// TwinCAT 3 PLC project Builder1
// ProgramVersion: 3.1.4023.0
// libraries:
//   Tc2_Standard, * (Beckhoff Automation GmbH)
//   Tc2_System, * (Beckhoff Automation GmbH)
//   Tc3_Module, * (Beckhoff Automation GmbH)
//   VisuSymbols,3.5.10.0,System
// project tree:
//   / Class Diagram.TcCD (not stored), ConcreteBuilder.TcPOU, Director.TcPOU, GlobalTextList.TcGTLO, ITF_Builder.TcIO, PlcTask.TcTTO, Product.TcPOU, Visualization Manager.TcVMO (not stored)
//   POUs/ MAIN.TcPOU
//   VISUs/ Visualization.TcVIS
// real-time tasks:
//   TASK PlcTask: cycle T#10ms, priority 20, ADS port 350

CONFIGURATION Builder1
    RESOURCE PLC ON TwinCAT3
        TASK PlcTask(INTERVAL := T#10ms, PRIORITY := 20);
        PROGRAM MAIN WITH PlcTask : MAIN;
    END_RESOURCE
END_CONFIGURATION

// ---- ITF_Builder.TcIO
///Builder interface to declare all needed parts to be built
INTERFACE ITF_Builder

///Illustrative method of the pattern to set the main part
METHOD Set_Main_Part
VAR_INPUT
	///Illustrative value (object because it is a TRING) to be set as a product part
	mainPart: STRING;
END_VAR
END_METHOD

///Illustrative method of the pattern to set the part1
METHOD Set_Part1
VAR_INPUT
	///Illustrative value (object because it is a TRING) to be set as a product part
	part1: STRING;
END_VAR
END_METHOD

///Illustrative method of the pattern to set the part2
METHOD Set_Part2
VAR_INPUT
	///Illustrative value (object because it is a TRING) to be set as a product part
	part2: STRING;
END_VAR
END_METHOD

///Illustrative method of the pattern to set the part3
METHOD Set_Part3
VAR_INPUT
	///Illustrative value (object because it is a TRING) to be set as a product part
	part3: STRING;
END_VAR
END_METHOD

END_INTERFACE

// ---- POUs/MAIN.TcPOU
PROGRAM MAIN
VAR
	///Three specifications arrays to be used by the same Director
	specsBuilder1: ARRAY[1..4] OF STRING := ['Red Chassis ', 'Sedan ', 'Motor 1.4cc ', 'Aluminium tires'];
	specsBuilder2: ARRAY[1..4] OF STRING := ['Black Chassis ', 'Hatchback ', 'Motor 2.0cc ', 'Chrome plated tires'];
	specsBuilder3: ARRAY[1..4] OF STRING := ['White Chassis ', 'Sport ', 'Motor 2.5cc ', 'Ligth aluminium tires'];
	///Special array for the visualization element
	tableArray: ARRAY[1..4, 1..3] OF STRING := ['Red Chassis', 'Black Chassis', 'White Chassis', 'Sedan', 'Hatchback', 'Sport', 'Motor 1.4cc', 'Motor 2.0cc', 'Motor 2.5cc', 'Aluminium tires', 'Chrome plated tires', 'Ligth aluminium tires'];
	///String variable to interact and respond to the client in the visualization element
	sMessageLog: STRING(500) := 'Waiting for your request';
	///Boolean value to react to a clients request
	bRequest: BOOL := FALSE;
	///Boolean and integer values to receive data from the tables in the visualization element
	///The boolean value validates if the client has chosen a valid option
	bRow: BOOL := FALSE;
	///The integer value hold the reference to the array of specifications
	iRow: INT := 0;
	///A pointer to Poduct to dynamically create and delete product objects at the clients requests
	prod: POINTER TO Product;
	///Three ConcreteBuilder instances to be passed to the Director and build the final Product objects
	///Each ConcreteBuilder intance is initiated with its own specifications
	{attribute 'old_input_assignments' := ''}
	concreteBuilder1: ConcreteBuilder(specs := specsBuilder1);
	{attribute 'old_input_assignments' := ''}
	concreteBuilder2: ConcreteBuilder(specs := specsBuilder2);
	{attribute 'old_input_assignments' := ''}
	concreteBuilder3: ConcreteBuilder(specs := specsBuilder3);
	///A Director instance that is instanciated with a ConcreteBuilder instance.
	/// later on in the program the specific ConcreteBuilder instance could be changed dynamically
	{attribute 'old_input_assignments' := ''}
	aDirector: Director(inputConcreteBuilder := concreteBuilder1);	
END_VAR

//The visualization element lets the client chose an option blueprint to build a Car
//Once the client has chosen his prefered option, he can then procede to make the request of construction.
//The bottom rectangle will handle all possible responses from te application to the client.

//If the client makes a request in the visualization element
IF bRequest
	THEN
	//CASE instruction to handle all possible cases of the cleint's request
	//The value to verify is iRow to specify which row the client has chosen
	CASE iRow OF
		//If the client has chosen the "Title" row from the visualization element we notify the client to chose a Car blueprint
		0: 	sMessageLog := 'You must first select a Car to make a request. Waiting for your request';
			//Once this reques has been handled, the reques flag is set to FALSE
			bRequest := FALSE;
		
		//If the client has chosen the first option row, the builder notifies the client about the received request
		1:	sMessageLog := 'Your red car is being built';
			//A new product object is created on demand
			prod := __NEW(Product);
			//The director object receives the ConcreteBuilder object to be used based on the clients choice
			aDirector(inputConcreteBuilder := concreteBuilder1);
			//The Product object request the construction to the Director.
			prod^ := aDirector.Construct();
			//The Builder's response after the Director object has handled the proper request
			sMessageLog := CONCAT( 'Your car has been built. It has ' , prod^.toString());
			//Once this reques has been handled, the reques flag is set to FALSE
			bRequest := FALSE;
			//Once this reques has been handled, the Product object is deleted to free memory
			__DELETE(prod);
			
		//If the client has chosen the second option row, the builder notifies the client about the received request	
		2:	sMessageLog := 'Your black car is being built';
			//A new product object is created on demand
			prod := __NEW(Product);
			//The director object receives the ConcreteBuilder object to be used based on the clients choice
			aDirector(inputConcreteBuilder := concreteBuilder2);
			//The Product object request the construction to the Director.
			prod^ := aDirector.Construct();
			//The Builder's response after the Director object has handled the proper request
			sMessageLog := CONCAT( 'Your car has been built. It has ' , prod^.toString());
			//Once this reques has been handled, the reques flag is set to FALSE
			bRequest := FALSE;
			//Once this reques has been handled, the Product object is deleted to free memory
			__DELETE(prod);
			
		//If the client has chosen the third option row, the builder notifies the client about the received request	
		3: sMessageLog := 'Your white car is being built';
			//A new product object is created on demand
			prod := __NEW(Product);
			//The director object receives the ConcreteBuilder object to be used based on the clients choice
			aDirector(inputConcreteBuilder := concreteBuilder3);
			//The Product object request the construction to the Director.
			prod^ := aDirector.Construct();
			//The Builder's response after the Director object has handled the proper request
			sMessageLog := CONCAT( 'Your car has been built. It has ' , prod^.toString());
			//Once this reques has been handled, the reques flag is set to FALSE
			bRequest := FALSE;
			//Once this reques has been handled, the Product object is deleted to free memory
			__DELETE(prod);
			
		//If the client makes any unrecognized request.	
		ELSE
			sMessageLog := 'That is not a valir selection. Waiting for your request';
			//Once this reques has been handled, the reques flag is set to FALSE
			bRequest := FALSE;

	END_CASE
END_IF

END_PROGRAM

// ---- Product.TcPOU
///The class Product is just a plain bluprint of the components of the object to be built.
///The final Product may ot may not contain the all the Parts listed on the Product declaration
/// rather only the parts in the specifications sent by the client.
{attribute 'enable_dynamic_creation' := ''}
FUNCTION_BLOCK Product
VAR_INPUT
	///List of possible parts to be build in a final Product object
	mainPart: STRING;
	part1: STRING;
	part2: STRING;
	part3: STRING;
END_VAR

///Method to be used in the visualization element for an easier String handling
METHOD toString : STRING
VAR
	///Local variable to join together and store the pieces of String
	tempString: STRING;
END_VAR
//tempString joins together "Main Part" and "Part 1" of the Product object
tempString := CONCAT(THIS^.mainPart , THIS^.part1);
//tempString joins together its current value and "Part 2" of the Product object
tempString := CONCAT(tempString , THIS^.part2);
//tempString joins together its current value and "Part 3" of the Product object
tempString := CONCAT(tempString , THIS^.part3);
//The final result is sent as the output of this method
toString := tempString;
END_METHOD

END_FUNCTION_BLOCK

// ---- ConcreteBuilder.TcPOU
///This is the concrete builder class, reponsible for building the final product object
FUNCTION_BLOCK ConcreteBuilder IMPLEMENTS ITF_Builder
VAR
	///Holds an internal reference to how the final product shoud be so the builder class can build it on the fly /// Contiene una referencia interna sobre cómo debe ser el producto final para que la clase constructora pueda construirlo sobre la marcha.
	/// without any help from other classes exepting the Director class that is going to be passing the special /// sin ninguna ayuda de otras clases excepto la clase Director que va a pasar el especial
	///specifications to the builder.///especificaciones para el constructor.
	localProduct: Product;
	///Stores the specifications, sent by the client, of the final product to be built.
	///Almacena las especificaciones, enviadas por el cliente, del producto final a construir.
	specifications: ARRAY[1..4] OF STRING;
END_VAR

METHOD fb_init
VAR_INPUT
	/// TRUE: the Retain-variables are initialized (reset warm / reset cold)
	bInitRetains: BOOL;
	/// TRUE  the instance will be copied to the copy-code afterward (online change)	
	bInCopyCode: BOOL;
	///The constructor receives the specifications for this ConcreteBuilder instance 
	///Just in case the concrete builder could change the specifications in the future, otherwise
	/// this specifications should be constant.
	specs: ARRAY[1..4] OF STRING;
END_VAR
//Stores the specifications on its own specifications field.
THIS^.specifications := specs;
END_METHOD

///Illustrative method of the pattern to get the main part
METHOD Get_Main_Part : STRING
//Returns the object stored in the built product THIS^.localProduct.mainPart
Get_Main_Part := THIS^.localProduct.mainPart;
END_METHOD

///Illustrative method of the pattern to get the part1
METHOD Get_Part1 : STRING
//Returns the object stored in the built product THIS^.localProduct.part1
Get_Part1 := THIS^.localProduct.part1;
END_METHOD

///Illustrative method of the pattern to get the part2
METHOD Get_Part2 : STRING
//Returns the object stored in the built product THIS^.localProduct.part2
Get_Part2 := THIS^.localProduct.part2;
END_METHOD

///Illustrative method of the pattern to get the part3
METHOD Get_Part3 : STRING
//Returns the object stored in the built product THIS^.localProduct.part3
Get_Part3 := THIS^.localProduct.part3;
END_METHOD

///Illustrative method of the pattern
METHOD Get_Result : Product
//The concrete builder, after it builts the final object of class product, returns the 
// final product object 
Get_Result := THIS^.localProduct;
END_METHOD

///Illustrative method of the pattern to set the main part
METHOD Set_Main_Part
VAR_INPUT
	///Illustrative value (object because it is a TRING) to be set as a product part
	mainPart: STRING;
END_VAR
//Sets the passed value to its corresponding field. 
//We can say that the the final product is in process of being built.
//So this is a step into building the final product done by the builder.
THIS^.localProduct.mainPart := mainPart;
END_METHOD

///Illustrative method of the pattern to set the part1
METHOD Set_Part1
VAR_INPUT
	///Illustrative value (object because it is a TRING) to be set as a product part
	part1: STRING;
END_VAR
//Sets the passed value to its corresponding field. 
//We can say that the the final product is in process of being built.
//So this is a step into building the final product done by the builder.
THIS^.localProduct.part1 := part1;
END_METHOD

///Illustrative method of the pattern to set the part2
METHOD Set_Part2
VAR_INPUT
	///Illustrative value (object because it is a TRING) to be set as a product part
	part2: STRING;
END_VAR
//Sets the passed value to its corresponding field. 
//We can say that the the final product is in process of being built.
//So this is a step into building the final product done by the builder.
THIS^.localProduct.part2 := part2;
END_METHOD

///Illustrative method of the pattern to set the part3
METHOD Set_Part3
VAR_INPUT
	///Illustrative value (object because it is a TRING) to be set as a product part
	part3: STRING;
END_VAR
//Sets the passed value to its corresponding field. 
//We can say that the the final product is in process of being built.
//So this is a step into building the final product done by the builder.
THIS^.localProduct.part3 := part3;
END_METHOD

END_FUNCTION_BLOCK

// ---- Director.TcPOU
///The director class is responsible to delegate the construction of the final product object 
/// to a concrete builder object.
{attribute 'enable_dynamic_creation' := ''}
FUNCTION_BLOCK Director
VAR_INPUT
	///Reference to the builder that is going to be building the final product object.
	///Referencia al constructor que construirá el objeto del producto final.
	{attribute 'old_input_assignments' := ''}
	inputConcreteBuilder: ConcreteBuilder(specs := inputConcreteBuilder.specifications);
END_VAR
VAR
	///Holds a reference to the concrete builder object to send the specifications of the final product to it.
	/// Contiene una referencia al objeto constructor concreto para enviarle las especificaciones del producto final
	{attribute 'old_input_assignments' := ''}
	concreteBuilder: ConcreteBuilder(specs := THIS^.concreteBuilder.specifications);
END_VAR

//Stores the reference to which builder will be building the final product object in its own field THIS^.concreteBuilder
//Almacena la referencia a qué constructor construirá el objeto del producto final en su propio campo THIS^.concreteBuilder
THIS^.concreteBuilder := inputConcreteBuilder;

///This method is going to be called by the client when a new Product object must be built
METHOD Construct : Product
//The Director tells its concreteBuilder instance to build the final product step by step passing the specifications stored in the 
// concreteBuilder array THIS^.specifications[1..4]

//Step 1 "Main Part"
THIS^.concreteBuilder.Set_Main_Part(THIS^.concreteBuilder.specifications[1]);
//Step 2 "Part 1"
THIS^.concreteBuilder.Set_Part1(THIS^.concreteBuilder.specifications[2]);
//Step 3 "Part 2"
THIS^.concreteBuilder.Set_Part2(THIS^.concreteBuilder.specifications[3]);
//Step 4 "Part 3"
THIS^.concreteBuilder.Set_Part3(THIS^.concreteBuilder.specifications[4]);

//Finally the concreteBuilder instance in the Director object delivers the final result as a Product object
//Finalmente, la instancia de concreteBuilder en el objeto Director entrega el resultado final como un objeto Producto
Construct := THIS^.concreteBuilder.Get_Result();
END_METHOD

///This constructor is called at instanciation it is necessary to instanciate the Director instance.
///The specifications of the concreteBuilder instance stored in the Director instance should be set first by the client
/// otherwise a Data Recursion error is caused
METHOD fb_init
VAR_INPUT
	/// TRUE: the Retain-variables are initialized (reset warm / reset cold)
	bInitRetains: BOOL;
	/// TRUE  the instance will be copied to the copy-code afterward (online change)
	bInCopyCode: BOOL;
	///Reference a concreteBuilder instance to instanciate the Director.
	{attribute 'old_input_assignments' := ''}
	inputConcreteBuilder: ConcreteBuilder(specs := defaultArray);
END_VAR
VAR
	///Variable to isntanciate the concreteBuilder instance on the input section. It does not affect the Directors instanciation.
	defaultArray: ARRAY[1..4] OF STRING := ['Default', 'Default', 'Default', 'Default'];
END_VAR
//Creates the concreteBuilder instance that will be building the final product object in its own field THIS^.concreteBuilder
//This instance is empty because we can not use Data Recursion with the inputConcreteInstance instanciation.
//So this concreteBuilder instance should be changed by the client before a Construct() request is called on the Director for the first time only.
THIS^.concreteBuilder := inputConcreteBuilder;
END_METHOD

END_FUNCTION_BLOCK

// ---- GlobalTextList.TcGTLO
TEXTLIST GlobalTextList
  801 = '%s'
  649 = 'Builder´s response'
  337 = 'Car type'
  930 = 'Chassis Colour'
  823 = 'choose Your new Car'
  637 = 'f'
  278 = 'Make Request'
  511 = 'Motor dimensions'
  584 = 'Wheels type'
END_TEXTLIST

// ---- VISUs/Visualization.TcVIS
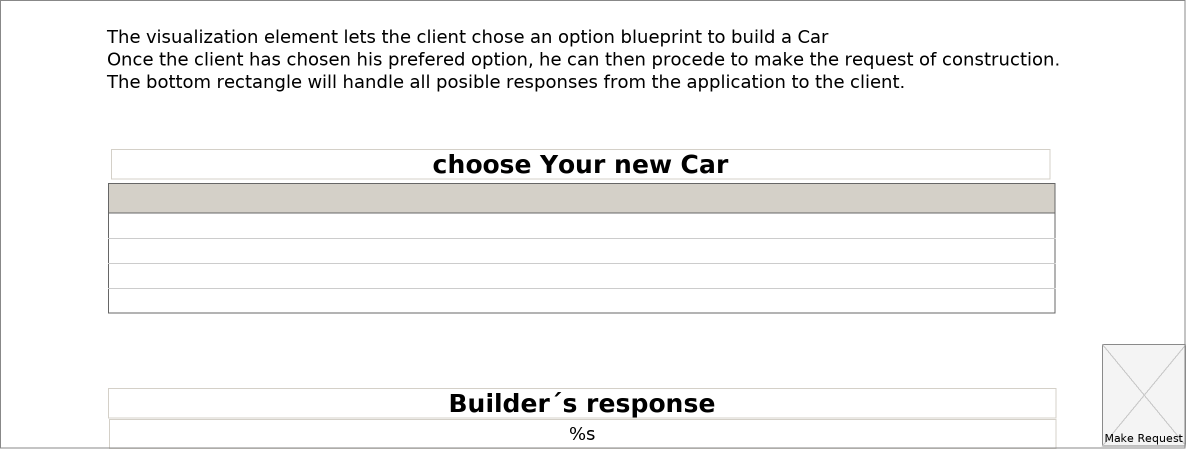
VISUALIZATION Visualization  // 1186x449
    Table (108,183 947x130), data array: MAIN.tableArray
        p3854506369: MAIN.tableArray[1,INDEX]
        p1892666644: MAIN.tableArray[2,INDEX]
        p338671338: MAIN.tableArray[3,INDEX]
        p2170511999: MAIN.tableArray[4,INDEX]
        p2232123230: Chassis Colour
        p511219082: Car type
        p1755163831: Motor dimensions
        p4092479075: Wheels type
        p1137915858: MAIN.iRow
        p1822360349: MAIN.bRow
    Textfield (111,149 939x30), "choose Your new Car"
    Textfield (108,388 948x30), "Builder´s response"
    Textfield (109,419 947x30), "%s", text variable: MAIN.sMessageLog
    Image (1102,344 84x102), "Make Request", image: VisuSymbols.Symbols.OK
        OnMouseClick: toggle MAIN.bRequest
    Label (104,10 953x99), "The visualization element lets the client chose an option blueprint to build a Car Once the client has chosen his prefered option, he can then procede to make the request of construction. The bottom rectangle will handle all posible responses from the application to the client."
END_VISUALIZATION
